{attribute 'qualified_only'}
//{attribute 'strict'}
{attribute 'to_string'}

TYPE E_Cluster_State_Cmd :
(
	Idle := 0,
	Warmup := 1,
	Cycling := 2,
	Shutdown := 3,
	Reset_Fault := 4
);
END_TYPE

(* stored: Version 1.1.0.1, ProductVersion 3.1.4024.12
   DUT E_Cluster_State_Cmd: Id {1b9102f1-1f0f-45a4-952d-da0fdfc2c421} *)
